SUBAPPLICATION NumericValue_PHYS_TO_INI (* Numerischer VT-Wert (PHYS-Variante, skaliert) einlesen und in INI speichern (generisch). *)
  (* Standard: 61499-2 *)
  (* Version 1.0, 2026-09-09, Franz Höpfinger, Meisterschulen am Ostbahnhof, Ausgelagert aus Uebung_012e_sub zur Wiederverwendung. *)
  PACKAGE MyLib::sys;
  IMPORT isobus::UT::Q::const::IDs::ID_NULL;
  IMPORT logiBUS::utils::conversion::phys::NumericObjectPool_S;
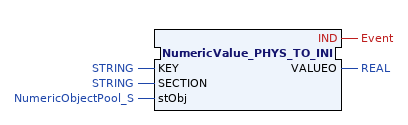
  EVENT_OUTPUT
    IND;
  END_EVENT
  VAR_INPUT
    KEY : STRING; (* Key name. *)
    SECTION : STRING; (* Section name. *)
    stObj : logiBUS::utils::conversion::phys::NumericObjectPool_S := (u16ObjId := ID_NULL, r32Scale := 1.0, i32Offset := 0, u8Decimals := 0);
  END_VAR
  VAR_OUTPUT
    VALUEO : REAL;
  END_VAR
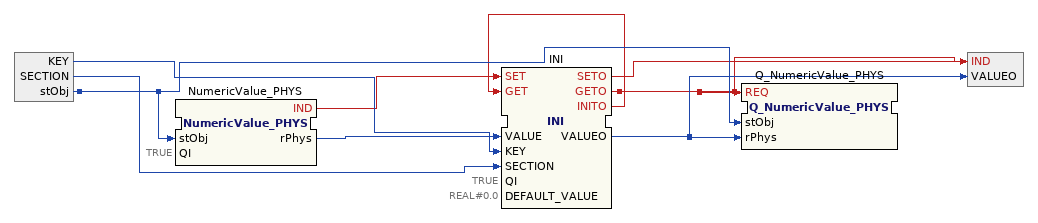
  FBS
    NumericValue_PHYS : isobus::UT::io::NumericValue::NumericValue_PHYS(QI := TRUE);
    INI : eclipse4diac::storage::INI(QI := TRUE, DEFAULT_VALUE := REAL#0.0);
    Q_NumericValue_PHYS : isobus::UT::Q::Q_NumericValue_PHYS;
  END_FBS
  EVENT_CONNECTIONS
    NumericValue_PHYS.IND TO INI.SET;
    INI.SETO TO IND;
    INI.GETO TO Q_NumericValue_PHYS.REQ;
    INI.GETO TO IND;
    INI.INITO TO INI.GET;
  END_CONNECTIONS
  DATA_CONNECTIONS
    NumericValue_PHYS.rPhys TO INI.VALUE;
    stObj TO Q_NumericValue_PHYS.stObj;
    KEY TO INI.KEY;
    INI.VALUEO TO Q_NumericValue_PHYS.rPhys;
    INI.VALUEO TO VALUEO;
    stObj TO NumericValue_PHYS.stObj;
    SECTION TO INI.SECTION;
  END_CONNECTIONS
END_SUBAPPLICATION
